FUNCTION_BLOCK CL_AxisMCMaster EXTENDS CL_AxisMC
VAR
  //objAxisDriver : CL_AxisDriverMaster; //Axis Master has no hardware driver
END_VAR

SUPER^();

METHOD PUBLIC Init : BOOL
VAR_INPUT
  stIrrLine       : ST_LineReference;
  stAxisMaster_P  : POINTER TO AXIS_REF;
END_VAR
Init := SUPER^.InitMC(stIrrLine := stIrrLine, stAxisMotor_P := stAxisMaster_P, stAxisMaster_P := stAxisMaster_P, AxisDriver_P := 0);
END_METHOD

METHOD PROTECTED InitDefect : BOOL
InitDefect := SUPER^.InitDefect();
ADSLOGSTR(ADSLOG_MSGTYPE_LOG, 'CL_AxisMCMaster init defect','');
END_METHOD

METHOD PROTECTED InitParams : BOOL
VAR_INPUT
END_VAR
InitParams := SUPER^.InitParams();
_sWhichAxis := 'virtual-master';
END_METHOD

END_FUNCTION_BLOCK

(* stored: Version 1.1.0.1, ProductVersion 3.1.4024.12
   POU CL_AxisMCMaster: Id {f408589f-d93f-4ed2-926a-1d5fc7672154}, SpecialFunc None
   Method Init: Id {554b1c05-cf3a-4a4b-8b69-f624e8441e8d}
   Method InitDefect: Id {66a7c3c9-7aff-4ac1-982c-d54ef8229c1c}
   Method InitParams: Id {37e7851f-c095-4029-91b1-33b5447071e8} *)
